FUNCTION TailEndianSwap : EspUdpEnd
VAR_INPUT
	In	: EspUdpEnd;
END_VAR
VAR
END_VAR

In.EndDelimiter			:= BE16_TO_HOST(In.EndDelimiter);

TailEndianSwap := In;

END_FUNCTION

(* stored: Version 1.1.0.1
   POU TailEndianSwap: Id {b83d4834-125c-4a8f-ba5a-f0b762aa00d5}, SpecialFunc None *)
